TYPE ST_CommandChangeMode :
STRUCT
	cmdChangeProduction	 	  	: FB_CommandChange;
	cmdChangeMaintenance		: FB_CommandChange;
	cmdChangeManual		    	: FB_CommandChange;
	cmdChangeWashing		   	: FB_CommandChange;
	cmdChangeDiagnostics		: FB_CommandChange;
END_STRUCT
END_TYPE

(* stored: Version 1.1.0.1
   DUT ST_CommandChangeMode: Id {b75752ec-7f06-0c94-055d-596f76bcbf81} *)
